Staubli VAL3: getType.pgx

public program getType(num& x_nType, bool x_bCycle, num x_nIndex)
begin
  // get the point Type
  if x_bCycle
    x_nType=pt:tTraj[sTrajCycle].tData[x_nIndex].nType
  else
    x_nType=pEditPoint.tData[x_nIndex].nType
  endIf
end
